TYPE ST_CommonData :
STRUCT
	itfLogger				: ITF_BaseLogger;
	itfTime					: ITF_BaseTime;
	itfLocaciotn			: ITF_BaseLocation;
END_STRUCT
END_TYPE

(* stored: Version 1.1.0.1
   DUT ST_CommonData: Id {cf0974a8-7b75-0485-0608-2eb2da826506} *)
